TYPE ST_FileDialogParams :
STRUCT
	sTitle 		: STRING;
	sDirectory 	: STRING(255);
	sFile 		: STRING(255);
	sFilter 	: STRING;
	bInit 		: BOOL;
END_STRUCT
END_TYPE

(* stored: Version 1.1.0.1, ProductVersion 3.1.4022.6
   DUT ST_FileDialogParams: Id {e8834879-be10-4256-a6da-1be357d434da} *)
